(* CoDeSys 2.3.9.47 project: bms2.pro *)
(* Libraries: SysLibSockets.lib 22.5.14 15:16:32, WagoCANLayer2_02.lib 23.6.14 12:08:28, Standard.lib 20.5.14 07:13:26, Iecsfc.lib 16.5.13 13:00:50, SYSLIBCALLBACK.LIB 16.5.13 13:00:50 *)

(* PLC configuration (modules and I/O channels)
K-Bus [K_Bus] node 0, in %IB0 out %QB0 {KbusBusMode = 1; KbusCycleTime = 10000; KbusThreadPriority = 0; KbusSetOutputsToZeroOnApplicationStop = 1}
Modbus variables [PFC200MODBUS] node 1, in %IB0 out %QB0 {PlcStopBehaviour = 1; FiledbusErrorBehaviour = 1; TcpOperation = 1; TcpPort = 502; TcpTimeout = 600; UdpOperation = 1; UdpPort = 502; RtuOperation = 0; NodeId = 1; ResponseTimeout = 5000; Interface = 0; Baud = 115200; StopBits = 1; Parity = 1; FlowCtrl = 0; PhysInterface = 0}
CAN Layer2 Device [PFC200CANLAYER2] node 2, in %IB6000 out %QB6000 {PFC200CanLayer2NONE = 0}
Modbus-Master [MB_MASTER] node 3, in %IB0 out %QB0
*)

(* Task configuration *)
TASK TMAIN (PRIORITY := 6, INTERVAL := T#100ms);
	PLC_PRG();
END_TASK

(* POU PLC_PRG, ST *)
 PROGRAM PLC_PRG
VAR
	canOpenPort : CAN_OPEN;
	xOpenPort : BOOL := TRUE;
	xPortIsOpen : BOOL;
	fbCanRecv : CAN_RX_11BIT_FRAME :=(
		 CAN_ID := 16#305,
		 CAN_BUFFER := FALSE );
	aRecvData : ARRAY [1..8] OF BYTE;
	bRecvLen : BYTE;

	recvDataFromId306  : CAN_RX_11BIT_FRAME := (
		CAN_ID := 16#0306,
		CAN_BUFFER := FALSE);
	recvData306 : ARRAY [1..8] OF BYTE;

	xRead : BOOL;

	fbCanSend			: CAN_TX_11BIT_FRAME :=(
		CAN_ID			:= 16#305,
		RTR_FRAME		:= FALSE,
		DATALENGTH	:= 8 );
	xWrite				: BOOL;
	aSendData			: ARRAY [1..8] OF BYTE; (* := 80, 0, 0, 0, 0, 0, 0, 0;*)
	tSend				: TON :=(PT:= t#10ms );

	data306				: ARRAY [1..8] OF BYTE;
	(*fbCanSend306			: CAN_TX_11BIT_FRAME :=(
		CAN_ID			:= 16#306,
		RTR_FRAME		:= FALSE,
		DATALENGTH	:= 8 );
	fbCanSend307			: CAN_TX_11BIT_FRAME :=(
		CAN_ID			:= 16#307,
		RTR_FRAME		:= FALSE,
		DATALENGTH	:= 8 );
	data307 				: ARRAY [1..8] OF BYTE := 62,6,64,49,62,6,64,49;*)


	(*mqttClient: MQTT_Client;
	xPublish : BOOL;
	xSubscribe : BOOL;*)
END_VAR
canOpenPort(BAUDRATE:= 500000, ENABLE:= xOpenPort);

fbCanRecv(
	 ENABLE := xPortIsOpen,
	 READ_FRAME := xRead );
recvDataFromId306(
	ENABLE := xPortIsOpen,
	 READ_FRAME := xRead );
fbCanSend(
	DATA:= aSendData,
	ENABLE:= xPortIsOpen,
	WRITE_FRAME:= xWrite );

(*fbCanSend306(
	DATA := data306,
	ENABLE := xPortIsOpen,
	WRITE_FRAME := xWrite
);
fbCanSend307(
	DATA := data307,
	ENABLE := xPortIsOpen,
	WRITE_FRAME := xWrite
);*)
IF canOpenPort.CONFIRM AND canOpenPort.ERROR = CAN_PORT_OK THEN
	 xOpenPort := FALSE;
	 xPortIsOpen := TRUE;
END_IF

tSend(IN := TRUE AND NOT xWrite);
IF tSend.Q THEN (* sending message *)
		tSend(IN := FALSE);
		xWrite := TRUE;
END_IF


IF xPortIsopen AND NOT xRead THEN
	 IF fbCanRecv.ERROR = CAN_RECEIVE_OK  THEN
		 aRecvData := fbCanRecv.DATA;
		 aSendData := aRecvData; (*16#305*)
		 (*recvData306 := canRecv306.DATA;
		 data306 := recvData306;
		 data306[4] := 1;*)
		 bRecvLen := fbCanRecv.DATALENGTH;
		 xRead := TRUE;
	 ELSE
		xRead := TRUE;
	 END_IF
END_IF


(*
mqttClient(
	sIp:= '10.210.10.60',
	wPortNumber:= 1883,
	sUsername:= '',
	sPassword:= '',
	xPublish:= xPublish, (* I/O variable to publish to a TOPIC *)
	xSubscribe:= xSubscribe (* NOT SUPPORTED, but must be here for I/O *)
 );

mqttClient.sTopic := 'ZAE/HOF/BMS/';
mqttClient.sPayload := BOOL_TO_STRING(FALSE);
xPublish := TRUE;
*)
END_PROGRAM
